{attribute addProperty BoxType "EP9214-0023-0019"}
{attribute addProperty Id "DPO_Inputs_ChannelAT %I*ARRAY[0..3] OF DPO_Inputs_Channel_A7741542320400DPO_Inputs_DeviceAT %I*DPO_Inputs_Device_A21D939180100DPO_Outputs_ChannelAT %Q*ARRAY[0..3] OF DPO_Outputs_Channel_5760563F128160DPO_Outputs_DeviceAT %Q*DPO_Outputs_Device_6EB864581620WcStateAT %I*WcState_F855686C1620InfoDataAT %I*InfoData_BC63D37F80100"}
{attribute addProperty CRC "466435085"}
{attribute addProperty SizeInBites "640"}
{attribute addProperty SizeInBytes "80"}
TYPE EP9214_38F98C76 :
STRUCT
	{attribute addProperty Name "DPO_Inputs_Channel"}
	DPO_Inputs_Channel : ARRAY[0..3] OF DPO_Inputs_Channel_A7741542;
	{attribute addProperty Name "DPO_Inputs_Device"}
	DPO_Inputs_Device : DPO_Inputs_Device_A21D9391;
	{attribute addProperty Name "DPO_Outputs_Channel"}
	DPO_Outputs_Channel : ARRAY[0..3] OF DPO_Outputs_Channel_5760563F;
	{attribute addProperty Name "DPO_Outputs_Device"}
	DPO_Outputs_Device : DPO_Outputs_Device_6EB86458;
	{attribute addProperty Name "WcState"}
	WcState : WcState_F855686C;
	{attribute addProperty Name "InfoData"}
	InfoData : InfoData_BC63D37F;
END_STRUCT
END_TYPE

(* stored: Version 1.2.0.0, ProductVersion 3.1.4024.9
   DUT EP9214_38F98C76: Id {b7468f6a-ffe4-4a85-8208-e5eeb1ff50ed} *)
